ABB RAPID module: TCP_tSpindleSensor.mod

MODULE TCP_tSpindleSensor
	! Points are read in order of declaration.
  ! Please do not change the order of points!

  LOCAL PERS robtarget pTCP_Point1:=[[-313.4051,-948.094,744.0695],[0.00273810233920813,-0.707533657550812,-0.00241054152138531,0.706670165061951],[-2,0,-1,0],[9E+09,9E+09,9E+09,9E+09,9E+09,9E+09]];
	LOCAL PERS robtarget pTCP_Point2:=[[-475.6021,-946.3951,718.8234],[0.00315442332066596,-0.826922357082367,-0.00188407022505999,0.562304079532623],[-2,0,-1,0],[9E+09,9E+09,9E+09,9E+09,9E+09,9E+09]];
	LOCAL PERS robtarget pTCP_Point3:=[[-508.1882,-964.5076,724.9991],[0.22367949783802,0.796088516712189,0.155937910079956,-0.540271997451782],[-2,0,0,0],[9E+09,9E+09,9E+09,9E+09,9E+09,9E+09]];
	LOCAL PERS robtarget pTCP_Point4:=[[-356.5605,-887.2413,735.593],[0.446088463068008,0.541921854019165,0.318820506334305,-0.636929512023926],[-2,-1,0,0],[9E+09,9E+09,9E+09,9E+09,9E+09,9E+09]];

ENDMODULE
